// TIA Portal V19 export
DATA_BLOCK "A0301_Fermi_P1"   // DB51
// stored: InstanceOfName A0301_Fermi_P1_FB, InstanceOfType FB
"A0301_Fermi_P1_FB"
   // VAR_INPUT
   //    AreaInterface : "AreaInterface";
   //    ZSI : "udt_ZoneSafetyInterface";
   //    DSI : "udt_DeviceSafetyInterface";
   //    DataIn : Struct
   //       OP_Rest_PB : Bool := FALSE;
   //       OP_Work_PB : Bool := FALSE;
   //    END_STRUCT;
   //    CIn : Struct
   //       Manager_Fermi : "ValveMachine_Manager";
   //       Manager_Paregg : "ValveMachine_Manager";
   //       SemiAut : Bool := FALSE;
   //       P1 : Struct
   //          Cndz_Sfalsatore : Bool := FALSE;
   //          Cndz_Pareggiatore : Bool := FALSE;
   //       END_STRUCT;
   //       Trasporto : "SpeedMachine_COut";
   //    END_STRUCT;
   //    Config : Struct
   //       Fermi : Array[1..6] of "ValveMachine_Config";
   //       Pareggiatore : "ValveMachine_Config";
   //       DelayMissingCondition : Time := T#3S;
   //    END_STRUCT;
   // END_VAR
   // VAR_OUTPUT
   //    MachineInterface : "MachineInterface";
   //    COut : Struct
   //       Fermi : "ValveMachine_COut";
   //       Pareggiatore : "ValveMachine_COut";
   //    END_STRUCT;
   // END_VAR
   // VAR
   //    Alarm : Struct
   //       Fermi : Array[1..6] of "ValveAlr";
   //       Pareggiatore { S7_SetPoint := 'True'} : "ValveAlr";
   //    END_STRUCT;
   //    Warning : Struct
   //       OP_REST_MissingCnd : Bool := FALSE;
   //       OP_WORK_MissingCnd : Bool := FALSE;
   //       Fermi : Array[1..6] of "ValveMachine_Wng";
   //       Pareggiatore { S7_SetPoint := 'True'} : "ValveMachine_Wng";
   //    END_STRUCT;
   //    HMI : Struct
   //       Selection : Array[1..6] of Bool;
   //       FermiSts { S7_SetPoint := 'True'} : "UDT_HMI-Sts_ValvePosA0301";
   //       PareggiatoreSts { S7_SetPoint := 'True'} : "UDT_HMI-Sts_ValvePosA0301";
   //       B_ResetShiftDone : Bool := FALSE;
   //    END_STRUCT;
   //    Sts : Struct
   //       Fermi_AlarmPresence : Bool := FALSE;
   //       OP_CanMoveFreely : Bool := TRUE;
   //       OP_Rest_Cnd : Bool := TRUE;
   //       Op_Work_Cnd : Bool := TRUE;
   //    END_STRUCT;
   //    Ctrl : Struct
   //       OP_Rest_Man : Bool := FALSE;
   //       OP_Work_Man : Bool := FALSE;
   //       OP_Rest_Aut : Bool := FALSE;
   //       OP_Work_Aut : Bool := FALSE;
   //       OP_Rest : Bool := FALSE;
   //       OP_Work : Bool := FALSE;
   //    END_STRUCT;
   //    Fermi : Array[1..6] of "ValveMachine_FB";
   //    Pareggiatore { S7_SetPoint := 'True'} : "ValveMachine_FB";
   //    AUX : Struct
   //       OP_Rest_PB : Bool := FALSE;
   //       OP_Work_PB : Bool := FALSE;
   //    END_STRUCT;
   //    TON_OP_REST_MissingCnd { S7_SetPoint := 'True'} : TON_TIME;
   //    TON_OP_WORK_MissingCnd { S7_SetPoint := 'True'} : TON_TIME;
   // END_VAR
BEGIN
   AreaInterface.EStop := FALSE;
   AreaInterface.Man := TRUE;
   AreaInterface.Aut := FALSE;
   AreaInterface.Cycle := FALSE;
   AreaInterface.StopInPhase := FALSE;
   AreaInterface.StopProgrammed := FALSE;
   AreaInterface.RstAlarms := FALSE;
   AreaInterface.ManOneShot := FALSE;
   AreaInterface.AutOneShot := FALSE;
   AreaInterface.CycleOneShot := FALSE;
   AreaInterface.CheckAutReady := FALSE;
   ZSI.Door_NormalStop := FALSE;
   ZSI.Door_SafeStop := FALSE;
   ZSI.Door_Opened := FALSE;
   ZSI.Door_EntryEnable := FALSE;
   DSI.SafeStop := FALSE;
   DSI.PowerEnable := TRUE;
   DSI.DevicesInSafeState := FALSE;
   CIn.Manager_Fermi.EnableStopDoorOpeningReq := FALSE;
   CIn.Manager_Fermi.EnableStopInPhase := FALSE;
   CIn.Manager_Fermi.EnableStopProgrammed := FALSE;
   CIn.Manager_Fermi.Control_ON := FALSE;
   CIn.Manager_Fermi.Rest := FALSE;
   CIn.Manager_Fermi.Work := FALSE;
   CIn.Trasporto.Infeed_ReqON := FALSE;
   CIn.Trasporto.CtrlSafe := FALSE;
   CIn.Trasporto.Standstill := TRUE;
   CIn.Trasporto.Bwd_CheckNext := FALSE;
   CIn.Trasporto.Fwd_CheckNext := FALSE;
   CIn.Trasporto.Bwd_VelZero := FALSE;
   CIn.Trasporto.Bwd_Running := FALSE;
   CIn.Trasporto.Fwd_VelZero := FALSE;
   CIn.Trasporto.Fwd_Running := FALSE;
   CIn.Trasporto.ActualVelocity := 0.0;
   CIn.Trasporto.TargetVelocity := 0.0;
   CIn.Trasporto.MaxVelocity := 39597.8;
   Config.Fermi[1..6].DelayPressureRunningTimeout := T#3S;
   Config.Fermi[1..6].DelayMissingCondition := T#3S;
   Config.Fermi[1..6].Rest_LsQty := 1;
   Config.Fermi[1..6].Work_LsQty := 0;
   Config.Fermi[1..6].Rest_RetainAut := FALSE;
   Config.Fermi[1..6].Work_RetainAut := FALSE;
   Config.Fermi[1..6].V.RestLimSwitchExist := TRUE;
   Config.Fermi[1..6].V.WorkLimSwitchExist := FALSE;
   Config.Fermi[1..6].V.CheckOilInPressure := FALSE;
   Config.Fermi[1..6].V.CutRestWhenIsAtRest := TRUE;
   Config.Fermi[1..6].V.CutWorkWhenIsAtWork := TRUE;
   Config.Fermi[1..6].V.RestTime := T#2S;
   Config.Fermi[1..6].V.WorkTime := T#2S;
   Config.Fermi[1..6].V.RestTimeOut := T#4S;
   Config.Fermi[1..6].V.WorkTimeOut := T#4S;
   Config.Pareggiatore.DelayPressureRunningTimeout := T#3S;
   Config.Pareggiatore.DelayMissingCondition := T#3S;
   Config.Pareggiatore.Rest_LsQty := 1;
   Config.Pareggiatore.Work_LsQty := 1;
   Config.Pareggiatore.Rest_RetainAut := FALSE;
   Config.Pareggiatore.Work_RetainAut := FALSE;
   Config.Pareggiatore.V.RestLimSwitchExist := TRUE;
   Config.Pareggiatore.V.WorkLimSwitchExist := TRUE;
   Config.Pareggiatore.V.CheckOilInPressure := FALSE;
   Config.Pareggiatore.V.CutRestWhenIsAtRest := TRUE;
   Config.Pareggiatore.V.CutWorkWhenIsAtWork := TRUE;
   Config.Pareggiatore.V.RestTime := T#1S;
   Config.Pareggiatore.V.WorkTime := T#1S;
   Config.Pareggiatore.V.RestTimeOut := T#1H;
   Config.Pareggiatore.V.WorkTimeOut := T#1H;
   MachineInterface.AutReady := FALSE;
   MachineInterface.Aborting := FALSE;
   MachineInterface.AckStopInPhase := FALSE;
   MachineInterface.AckStopProgrammed := FALSE;
   MachineInterface.MotionsStandStill := TRUE;
   MachineInterface.AlarmsPresence := FALSE;
   MachineInterface.WarningPresence := FALSE;
   COut.Fermi.CtrlSafe := FALSE;
   COut.Fermi.Standstill := TRUE;
   COut.Fermi.ReqOilPressure := FALSE;
   COut.Fermi.Rest_CheckNext := FALSE;
   COut.Fermi.Work_CheckNext := FALSE;
   COut.Fermi.Rest := FALSE;
   COut.Fermi.Work := FALSE;
   COut.Pareggiatore.CtrlSafe := FALSE;
   COut.Pareggiatore.Standstill := TRUE;
   COut.Pareggiatore.ReqOilPressure := FALSE;
   COut.Pareggiatore.Rest_CheckNext := FALSE;
   COut.Pareggiatore.Work_CheckNext := FALSE;
   COut.Pareggiatore.Rest := FALSE;
   COut.Pareggiatore.Work := FALSE;
   Alarm.Fermi[1..6].TimeOutRest := FALSE;
   Alarm.Fermi[1..6].TimeOutWork := FALSE;
   Alarm.Fermi[1..6].LimitSwitches := FALSE;
   Alarm.Pareggiatore.TimeOutRest := FALSE;
   Alarm.Pareggiatore.TimeOutWork := FALSE;
   Alarm.Pareggiatore.LimitSwitches := FALSE;
   Warning.Fermi[1..6].NotAutReady := FALSE;
   Warning.Fermi[1..6].PressureRunning_Timeout := FALSE;
   Warning.Fermi[1..6].Rest_MissingExtEnable := FALSE;
   Warning.Fermi[1..6].Work_MissingExtEnable := FALSE;
   Warning.Fermi[1].Missing_Rest_Ls_ON[1..8] := FALSE;
   Warning.Fermi[2].Missing_Rest_Ls_ON[1..8] := FALSE;
   Warning.Fermi[3].Missing_Rest_Ls_ON[1..8] := FALSE;
   Warning.Fermi[4].Missing_Rest_Ls_ON[1..8] := FALSE;
   Warning.Fermi[5].Missing_Rest_Ls_ON[1..8] := FALSE;
   Warning.Fermi[6].Missing_Rest_Ls_ON[1..8] := FALSE;
   Warning.Fermi[1].Missing_Work_Ls_ON[1..8] := FALSE;
   Warning.Fermi[2].Missing_Work_Ls_ON[1..8] := FALSE;
   Warning.Fermi[3].Missing_Work_Ls_ON[1..8] := FALSE;
   Warning.Fermi[4].Missing_Work_Ls_ON[1..8] := FALSE;
   Warning.Fermi[5].Missing_Work_Ls_ON[1..8] := FALSE;
   Warning.Fermi[6].Missing_Work_Ls_ON[1..8] := FALSE;
   Warning.Pareggiatore.NotAutReady := FALSE;
   Warning.Pareggiatore.PressureRunning_Timeout := FALSE;
   Warning.Pareggiatore.Rest_MissingExtEnable := FALSE;
   Warning.Pareggiatore.Work_MissingExtEnable := FALSE;
   Warning.Pareggiatore.Missing_Rest_Ls_ON[1..8] := FALSE;
   Warning.Pareggiatore.Missing_Work_Ls_ON[1..8] := FALSE;
   HMI.Selection[1..6] := TRUE;
   HMI.FermiSts.Standstill := TRUE;
   HMI.FermiSts.Rest := FALSE;
   HMI.FermiSts.Work := FALSE;
   HMI.FermiSts.AlarmPresence := FALSE;
   HMI.PareggiatoreSts.Standstill := TRUE;
   HMI.PareggiatoreSts.Rest := FALSE;
   HMI.PareggiatoreSts.Work := FALSE;
   HMI.PareggiatoreSts.AlarmPresence := FALSE;
   Fermi[1..6].AreaInterface.EStop := FALSE;
   Fermi[1..6].AreaInterface.Man := TRUE;
   Fermi[1..6].AreaInterface.Aut := FALSE;
   Fermi[1..6].AreaInterface.Cycle := FALSE;
   Fermi[1..6].AreaInterface.StopInPhase := FALSE;
   Fermi[1..6].AreaInterface.StopProgrammed := FALSE;
   Fermi[1..6].AreaInterface.RstAlarms := FALSE;
   Fermi[1..6].AreaInterface.ManOneShot := FALSE;
   Fermi[1..6].AreaInterface.AutOneShot := FALSE;
   Fermi[1..6].AreaInterface.CycleOneShot := FALSE;
   Fermi[1..6].AreaInterface.CheckAutReady := FALSE;
   Fermi[1..6].ZSI.Door_NormalStop := FALSE;
   Fermi[1..6].ZSI.Door_SafeStop := FALSE;
   Fermi[1..6].ZSI.Door_Opened := FALSE;
   Fermi[1..6].ZSI.Door_EntryEnable := FALSE;
   Fermi[1..6].DSI.SafeStop := FALSE;
   Fermi[1..6].DSI.PowerEnable := TRUE;
   Fermi[1..6].DSI.DevicesInSafeState := FALSE;
   Fermi[1..6].DataIn.PB.Rest := FALSE;
   Fermi[1..6].DataIn.PB.Work := FALSE;
   Fermi[1..6].DataIn.PB.StartStop := FALSE;
   Fermi[1].DataIn.Rest_Ls[1] := TRUE;
   Fermi[1].DataIn.Rest_Ls[2..8] := FALSE;
   Fermi[2].DataIn.Rest_Ls[1] := TRUE;
   Fermi[2].DataIn.Rest_Ls[2..8] := FALSE;
   Fermi[3].DataIn.Rest_Ls[1] := TRUE;
   Fermi[3].DataIn.Rest_Ls[2..8] := FALSE;
   Fermi[4].DataIn.Rest_Ls[1] := TRUE;
   Fermi[4].DataIn.Rest_Ls[2..8] := FALSE;
   Fermi[5].DataIn.Rest_Ls[1] := TRUE;
   Fermi[5].DataIn.Rest_Ls[2..8] := FALSE;
   Fermi[6].DataIn.Rest_Ls[1] := TRUE;
   Fermi[6].DataIn.Rest_Ls[2..8] := FALSE;
   Fermi[1].DataIn.Work_Ls[1..8] := FALSE;
   Fermi[2].DataIn.Work_Ls[1..8] := FALSE;
   Fermi[3].DataIn.Work_Ls[1..8] := FALSE;
   Fermi[4].DataIn.Work_Ls[1..8] := FALSE;
   Fermi[5].DataIn.Work_Ls[1..8] := FALSE;
   Fermi[6].DataIn.Work_Ls[1..8] := FALSE;
   Fermi[1..6].Cin.Manager.EnableStopDoorOpeningReq := FALSE;
   Fermi[1..6].Cin.Manager.EnableStopInPhase := FALSE;
   Fermi[1..6].Cin.Manager.EnableStopProgrammed := FALSE;
   Fermi[1..6].Cin.Manager.Control_ON := FALSE;
   Fermi[1..6].Cin.Manager.Rest := FALSE;
   Fermi[1..6].Cin.Manager.Work := FALSE;
   Fermi[1..6].Cin.PressureRunning := FALSE;
   Fermi[1..6].Cin.Rest_ExtEnable := TRUE;
   Fermi[1..6].Cin.Work_ExtEnable := TRUE;
   Fermi[1..6].Cin.ExternalAlarms := FALSE;
   Fermi[1..6].Config.DelayPressureRunningTimeout := T#3S;
   Fermi[1..6].Config.DelayMissingCondition := T#3S;
   Fermi[1..6].Config.Rest_LsQty := 1;
   Fermi[1..6].Config.Work_LsQty := 0;
   Fermi[1..6].Config.Rest_RetainAut := FALSE;
   Fermi[1..6].Config.Work_RetainAut := FALSE;
   Fermi[1..6].Config.V.RestLimSwitchExist := TRUE;
   Fermi[1..6].Config.V.WorkLimSwitchExist := FALSE;
   Fermi[1..6].Config.V.CheckOilInPressure := FALSE;
   Fermi[1..6].Config.V.CutRestWhenIsAtRest := TRUE;
   Fermi[1..6].Config.V.CutWorkWhenIsAtWork := TRUE;
   Fermi[1..6].Config.V.RestTime := T#2S;
   Fermi[1..6].Config.V.WorkTime := T#2S;
   Fermi[1..6].Config.V.RestTimeOut := T#4S;
   Fermi[1..6].Config.V.WorkTimeOut := T#4S;
   Fermi[1..6].MachineInterface.AutReady := FALSE;
   Fermi[1..6].MachineInterface.Aborting := FALSE;
   Fermi[1..6].MachineInterface.AckStopInPhase := FALSE;
   Fermi[1..6].MachineInterface.AckStopProgrammed := FALSE;
   Fermi[1..6].MachineInterface.MotionsStandStill := TRUE;
   Fermi[1..6].MachineInterface.AlarmsPresence := FALSE;
   Fermi[1..6].MachineInterface.WarningPresence := FALSE;
   Fermi[1..6].COut.CtrlSafe := FALSE;
   Fermi[1..6].COut.Standstill := TRUE;
   Fermi[1..6].COut.ReqOilPressure := FALSE;
   Fermi[1..6].COut.Rest_CheckNext := FALSE;
   Fermi[1..6].COut.Work_CheckNext := FALSE;
   Fermi[1..6].COut.Rest := TRUE;
   Fermi[1..6].COut.Work := FALSE;
   Fermi[1..6].DataOut.RestSolenoid := FALSE;
   Fermi[1..6].DataOut.WorkSolenoid := FALSE;
   Fermi[1..6].Sts.Standstill := TRUE;
   Fermi[1..6].Sts.AlarmsPresence := FALSE;
   Fermi[1..6].Sts.WarningsPresence := FALSE;
   Fermi[1..6].Sts.Rest_Cnd := TRUE;
   Fermi[1..6].Sts.Work_Cnd := TRUE;
   Fermi[1..6].Ctrl.StopDueDoorOpeningRequest := FALSE;
   Fermi[1..6].Ctrl.StopInPhase := FALSE;
   Fermi[1..6].Ctrl.StopProgrammed := FALSE;
   Fermi[1..6].Ctrl.StopAborting := FALSE;
   Fermi[1..6].Ctrl.Work := FALSE;
   Fermi[1..6].Ctrl.Rest := FALSE;
   Fermi[1..6].Ctrl.Rest_Man := FALSE;
   Fermi[1..6].Ctrl.Work_Man := FALSE;
   Fermi[1..6].Ctrl.Rest_Aut := FALSE;
   Fermi[1..6].Ctrl.Work_Aut := FALSE;
   Fermi[1..6].V.ValveCtrl.SafeStop := FALSE;
   Fermi[1..6].V.ValveCtrl.Rst := FALSE;
   Fermi[1..6].V.ValveCtrl.MoveRest := FALSE;
   Fermi[1..6].V.ValveCtrl.MoveWork := FALSE;
   Fermi[1..6].V.RestLimitSwitch := TRUE;
   Fermi[1..6].V.WorkLimitSwitch := FALSE;
   Fermi[1..6].V.OilInPressure := FALSE;
   Fermi[1..6].V.Simulation := FALSE;
   Fermi[1..6].V.Config.RestLimSwitchExist := TRUE;
   Fermi[1..6].V.Config.WorkLimSwitchExist := FALSE;
   Fermi[1..6].V.Config.CheckOilInPressure := FALSE;
   Fermi[1..6].V.Config.CutRestWhenIsAtRest := TRUE;
   Fermi[1..6].V.Config.CutWorkWhenIsAtWork := TRUE;
   Fermi[1..6].V.Config.RestTime := T#2S;
   Fermi[1..6].V.Config.WorkTime := T#2S;
   Fermi[1..6].V.Config.RestTimeOut := T#4S;
   Fermi[1..6].V.Config.WorkTimeOut := T#4S;
   Fermi[1..6].V.ValveSts.AlarmPresence := FALSE;
   Fermi[1..6].V.ValveSts.RestPermit := TRUE;
   Fermi[1..6].V.ValveSts.RestInProgress := FALSE;
   Fermi[1..6].V.ValveSts.IsAtRest := TRUE;
   Fermi[1..6].V.ValveSts.WorkPermit := TRUE;
   Fermi[1..6].V.ValveSts.WorkInProgress := FALSE;
   Fermi[1..6].V.ValveSts.IsAtWork := FALSE;
   Fermi[1..6].V.ValveSts.StandStill := TRUE;
   Fermi[1..6].V.RestSolenoid := FALSE;
   Fermi[1..6].V.WorkSolenoid := FALSE;
   Fermi[1..6].V.ReqOilPressure := FALSE;
   Fermi[1..6].V.IsAtRest := TRUE;
   Fermi[1..6].V.IsAtWork := FALSE;
   Fermi[1..6].V.Ctrl.RestReq := FALSE;
   Fermi[1..6].V.Ctrl.WorkReq := FALSE;
   Fermi[1..6].V.Ctrl.RestSolenoid := FALSE;
   Fermi[1..6].V.Ctrl.WorkSolenoid := FALSE;
   Fermi[1..6].V.tonRest.PT := T#2S;
   Fermi[1..6].V.tonRest.IN := TRUE;
   Fermi[1..6].V.tonWork.PT := T#0MS;
   Fermi[1..6].V.tonWork.IN := FALSE;
   Fermi[1..6].V.tonTimeOutRest.PT := T#0MS;
   Fermi[1..6].V.tonTimeOutRest.IN := FALSE;
   Fermi[1..6].V.tonTimeOutWork.PT := T#0MS;
   Fermi[1..6].V.tonTimeOutWork.IN := FALSE;
   Fermi[1..6].TON_NoPendingCmd.PT := T#500MS;
   Fermi[1..6].TON_NoPendingCmd.IN := TRUE;
   Fermi[1..6].TON_Rest_MissingExtEnable.PT := T#0MS;
   Fermi[1..6].TON_Rest_MissingExtEnable.IN := FALSE;
   Fermi[1..6].TON_Work_MissingExtEnable.PT := T#0MS;
   Fermi[1..6].TON_Work_MissingExtEnable.IN := FALSE;
   Fermi[1..6].TON_PressureRunning_Timeout.PT := T#0MS;
   Fermi[1..6].TON_PressureRunning_Timeout.IN := FALSE;
   Fermi[1..6].Aux.Pb_Rest := FALSE;
   Fermi[1..6].Aux.Pb_Work := FALSE;
   Fermi[1..6].Aux.Pb_StartStop := FALSE;
   Pareggiatore.AreaInterface.EStop := FALSE;
   Pareggiatore.AreaInterface.Man := TRUE;
   Pareggiatore.AreaInterface.Aut := FALSE;
   Pareggiatore.AreaInterface.Cycle := FALSE;
   Pareggiatore.AreaInterface.StopInPhase := FALSE;
   Pareggiatore.AreaInterface.StopProgrammed := FALSE;
   Pareggiatore.AreaInterface.RstAlarms := FALSE;
   Pareggiatore.AreaInterface.ManOneShot := FALSE;
   Pareggiatore.AreaInterface.AutOneShot := FALSE;
   Pareggiatore.AreaInterface.CycleOneShot := FALSE;
   Pareggiatore.AreaInterface.CheckAutReady := FALSE;
   Pareggiatore.ZSI.Door_NormalStop := FALSE;
   Pareggiatore.ZSI.Door_SafeStop := FALSE;
   Pareggiatore.ZSI.Door_Opened := FALSE;
   Pareggiatore.ZSI.Door_EntryEnable := FALSE;
   Pareggiatore.DSI.SafeStop := FALSE;
   Pareggiatore.DSI.PowerEnable := TRUE;
   Pareggiatore.DSI.DevicesInSafeState := FALSE;
   Pareggiatore.DataIn.PB.Rest := FALSE;
   Pareggiatore.DataIn.PB.Work := FALSE;
   Pareggiatore.DataIn.PB.StartStop := FALSE;
   Pareggiatore.DataIn.Rest_Ls[1..8] := FALSE;
   Pareggiatore.DataIn.Work_Ls[1..8] := FALSE;
   Pareggiatore.Cin.Manager.EnableStopDoorOpeningReq := FALSE;
   Pareggiatore.Cin.Manager.EnableStopInPhase := FALSE;
   Pareggiatore.Cin.Manager.EnableStopProgrammed := FALSE;
   Pareggiatore.Cin.Manager.Control_ON := FALSE;
   Pareggiatore.Cin.Manager.Rest := FALSE;
   Pareggiatore.Cin.Manager.Work := FALSE;
   Pareggiatore.Cin.PressureRunning := FALSE;
   Pareggiatore.Cin.Rest_ExtEnable := TRUE;
   Pareggiatore.Cin.Work_ExtEnable := TRUE;
   Pareggiatore.Cin.ExternalAlarms := FALSE;
   Pareggiatore.Config.DelayPressureRunningTimeout := T#3S;
   Pareggiatore.Config.DelayMissingCondition := T#3S;
   Pareggiatore.Config.Rest_LsQty := 1;
   Pareggiatore.Config.Work_LsQty := 1;
   Pareggiatore.Config.Rest_RetainAut := FALSE;
   Pareggiatore.Config.Work_RetainAut := FALSE;
   Pareggiatore.Config.V.RestLimSwitchExist := TRUE;
   Pareggiatore.Config.V.WorkLimSwitchExist := TRUE;
   Pareggiatore.Config.V.CheckOilInPressure := FALSE;
   Pareggiatore.Config.V.CutRestWhenIsAtRest := TRUE;
   Pareggiatore.Config.V.CutWorkWhenIsAtWork := TRUE;
   Pareggiatore.Config.V.RestTime := T#1S;
   Pareggiatore.Config.V.WorkTime := T#1S;
   Pareggiatore.Config.V.RestTimeOut := T#1H;
   Pareggiatore.Config.V.WorkTimeOut := T#1H;
   Pareggiatore.MachineInterface.AutReady := FALSE;
   Pareggiatore.MachineInterface.Aborting := FALSE;
   Pareggiatore.MachineInterface.AckStopInPhase := FALSE;
   Pareggiatore.MachineInterface.AckStopProgrammed := FALSE;
   Pareggiatore.MachineInterface.MotionsStandStill := TRUE;
   Pareggiatore.MachineInterface.AlarmsPresence := FALSE;
   Pareggiatore.MachineInterface.WarningPresence := FALSE;
   Pareggiatore.COut.CtrlSafe := FALSE;
   Pareggiatore.COut.Standstill := TRUE;
   Pareggiatore.COut.ReqOilPressure := FALSE;
   Pareggiatore.COut.Rest_CheckNext := FALSE;
   Pareggiatore.COut.Work_CheckNext := FALSE;
   Pareggiatore.COut.Rest := FALSE;
   Pareggiatore.COut.Work := FALSE;
   Pareggiatore.DataOut.RestSolenoid := FALSE;
   Pareggiatore.DataOut.WorkSolenoid := FALSE;
   Pareggiatore.Sts.Standstill := TRUE;
   Pareggiatore.Sts.AlarmsPresence := FALSE;
   Pareggiatore.Sts.WarningsPresence := FALSE;
   Pareggiatore.Sts.Rest_Cnd := TRUE;
   Pareggiatore.Sts.Work_Cnd := TRUE;
   Pareggiatore.Ctrl.StopDueDoorOpeningRequest := FALSE;
   Pareggiatore.Ctrl.StopInPhase := FALSE;
   Pareggiatore.Ctrl.StopProgrammed := FALSE;
   Pareggiatore.Ctrl.StopAborting := FALSE;
   Pareggiatore.Ctrl.Work := FALSE;
   Pareggiatore.Ctrl.Rest := FALSE;
   Pareggiatore.Ctrl.Rest_Man := FALSE;
   Pareggiatore.Ctrl.Work_Man := FALSE;
   Pareggiatore.Ctrl.Rest_Aut := FALSE;
   Pareggiatore.Ctrl.Work_Aut := FALSE;
   Pareggiatore.V.ValveCtrl.SafeStop := FALSE;
   Pareggiatore.V.ValveCtrl.Rst := FALSE;
   Pareggiatore.V.ValveCtrl.MoveRest := FALSE;
   Pareggiatore.V.ValveCtrl.MoveWork := FALSE;
   Pareggiatore.V.RestLimitSwitch := FALSE;
   Pareggiatore.V.WorkLimitSwitch := FALSE;
   Pareggiatore.V.OilInPressure := FALSE;
   Pareggiatore.V.Simulation := FALSE;
   Pareggiatore.V.Config.RestLimSwitchExist := TRUE;
   Pareggiatore.V.Config.WorkLimSwitchExist := TRUE;
   Pareggiatore.V.Config.CheckOilInPressure := FALSE;
   Pareggiatore.V.Config.CutRestWhenIsAtRest := TRUE;
   Pareggiatore.V.Config.CutWorkWhenIsAtWork := TRUE;
   Pareggiatore.V.Config.RestTime := T#1S;
   Pareggiatore.V.Config.WorkTime := T#1S;
   Pareggiatore.V.Config.RestTimeOut := T#1H;
   Pareggiatore.V.Config.WorkTimeOut := T#1H;
   Pareggiatore.V.ValveSts.AlarmPresence := FALSE;
   Pareggiatore.V.ValveSts.RestPermit := TRUE;
   Pareggiatore.V.ValveSts.RestInProgress := FALSE;
   Pareggiatore.V.ValveSts.IsAtRest := FALSE;
   Pareggiatore.V.ValveSts.WorkPermit := TRUE;
   Pareggiatore.V.ValveSts.WorkInProgress := FALSE;
   Pareggiatore.V.ValveSts.IsAtWork := FALSE;
   Pareggiatore.V.ValveSts.StandStill := TRUE;
   Pareggiatore.V.RestSolenoid := FALSE;
   Pareggiatore.V.WorkSolenoid := FALSE;
   Pareggiatore.V.ReqOilPressure := FALSE;
   Pareggiatore.V.IsAtRest := FALSE;
   Pareggiatore.V.IsAtWork := FALSE;
   Pareggiatore.V.Ctrl.RestReq := FALSE;
   Pareggiatore.V.Ctrl.WorkReq := FALSE;
   Pareggiatore.V.Ctrl.RestSolenoid := FALSE;
   Pareggiatore.V.Ctrl.WorkSolenoid := FALSE;
   Pareggiatore.V.tonRest.PT := T#0MS;
   Pareggiatore.V.tonRest.IN := FALSE;
   Pareggiatore.V.tonWork.PT := T#0MS;
   Pareggiatore.V.tonWork.IN := FALSE;
   Pareggiatore.V.tonTimeOutRest.PT := T#0MS;
   Pareggiatore.V.tonTimeOutRest.IN := FALSE;
   Pareggiatore.V.tonTimeOutWork.PT := T#0MS;
   Pareggiatore.V.tonTimeOutWork.IN := FALSE;
   Pareggiatore.TON_NoPendingCmd.PT := T#500MS;
   Pareggiatore.TON_NoPendingCmd.IN := TRUE;
   Pareggiatore.TON_Rest_MissingExtEnable.PT := T#0MS;
   Pareggiatore.TON_Rest_MissingExtEnable.IN := FALSE;
   Pareggiatore.TON_Work_MissingExtEnable.PT := T#0MS;
   Pareggiatore.TON_Work_MissingExtEnable.IN := FALSE;
   Pareggiatore.TON_PressureRunning_Timeout.PT := T#0MS;
   Pareggiatore.TON_PressureRunning_Timeout.IN := FALSE;
   Pareggiatore.Aux.Pb_Rest := FALSE;
   Pareggiatore.Aux.Pb_Work := FALSE;
   Pareggiatore.Aux.Pb_StartStop := FALSE;
   TON_OP_REST_MissingCnd.PT := T#0MS;
   TON_OP_REST_MissingCnd.IN := FALSE;
   TON_OP_WORK_MissingCnd.PT := T#0MS;
   TON_OP_WORK_MissingCnd.IN := FALSE;
END_DATA_BLOCK
